(* Schneider Machine Expert - Basic project Memory bits S&P, file version 2.0.0.0 *)
(* ProjectInformations: Name=New project *)

HARDWARE
  Cpu 0: TM221CE16R
  EthernetConfiguration: NetworkName=M221, IpAllocationMode=FixedAddress, IpAddress=0.0.0.0, SubnetMask=0.0.0.0
  SerialLineConfiguration: Baud=Baud19200, Parity=ParityEven, DataBits=DataBits8, StopBits=StopBits1, PhysicalMedium=PhysicalMediumRs485, TransmissionMode=TransmissionModeModbusRtu, SlaveId=1, Addressing=SlaveAddressing
  MastTask: UsePeriodScanMode=false, PeriodScan=100
  FastTask: Period=255
  CpuBehavior: StartingMode=StartAsPreviousState, AutoSaveRamOnEeprom=true, WatchdogPeriod=250

SYMBOLS  (address, symbol, comment, settings)

POU New POU
  (* SectionNumber=1 *)

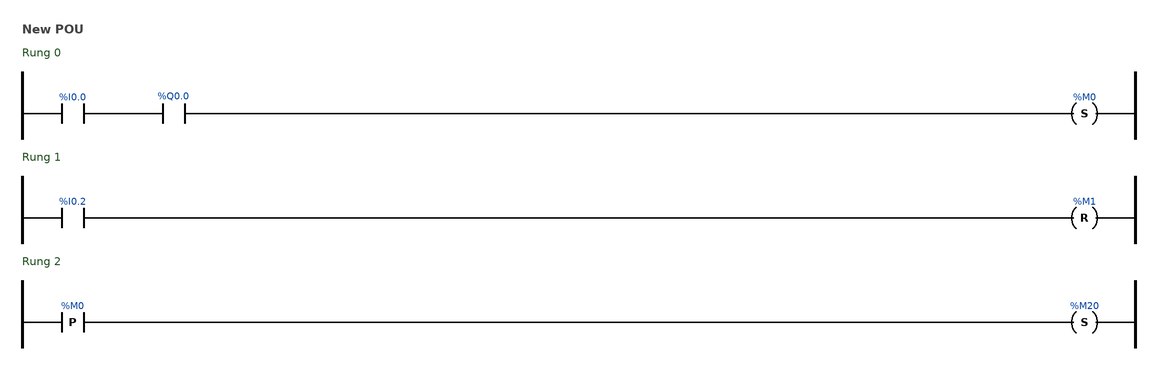

// Rung 0
  LD %I0.0
  AND %Q0.0
  S %M0
  // as ST:
  //   IF %I0.0 AND %Q0.0 THEN %M0 := TRUE; END_IF;

// Rung 1
  LD %I0.2
  R %M1
  // as ST:
  //   IF %I0.2 THEN %M1 := FALSE; END_IF;

// Rung 2
  LDR %M0
  S %M20
  // as ST:
  //   IF RISING(%M0) THEN %M20 := TRUE; END_IF;
